// TIA Portal V17 export
// export: Created 2024-09-02T12:49:55.2454988Z, ExportSetting WithDefaults, DisplayName Totally Integrated Automation Portal, DisplayVersion V17, DisplayName TIA Portal Openness, DisplayVersion V17, DisplayName TIA Portal Version Control Interface, DisplayVersion V17, DisplayName STEP 7 Professional, DisplayVersion V17, DisplayName STEP 7 Safety, DisplayVersion V17, DisplayName WinCC Professional, DisplayVersion V17
FUNCTION "SysFC_NumOfElementArray" : Void   // FC129, LAD
TITLE = Determining the number of elements in the array / Anzahl Elemente im Array ermitteln
{ S7_Optimized_Access := 'TRUE' }
AUTHOR : OlegFuehrus
FAMILY : DIAG
NAME : DIAG
VERSION : 0.1
// stored: AutoNumber true, IsIECCheckEnabled false, SetENOAutomatically false, UDAEnableTagReadback false
   VAR_INPUT
      Data : Variant;
   END_VAR
   VAR_OUTPUT
      NumOfElemets : UDInt;
      Fault : Bool;
   END_VAR
   VAR_TEMP
      t_VKE0 : Bool;
      t_VKE1 : Bool;
      t_Amount : UDInt;
      t_Fault : Bool;
   END_VAR
BEGIN

REGION Network 1: VKE0/1
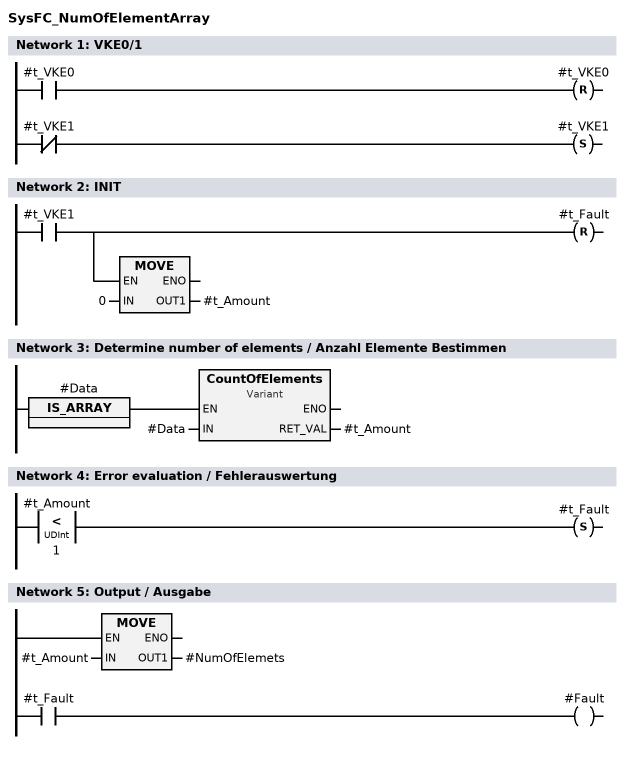
   RUNG wire#powerrail
      Contact( #t_VKE0 )
      R_Coil( #t_VKE0 )
   END_RUNG
   RUNG wire#powerrail
      I_Contact( #t_VKE1 )
      S_Coil( #t_VKE1 )
   END_RUNG
   // the same network as SCL:
   IF #t_VKE0 THEN #t_VKE0 := FALSE; END_IF;
   IF NOT #t_VKE1 THEN #t_VKE1 := TRUE; END_IF;
END_REGION

REGION Network 2: INIT
   RUNG wire#powerrail
      Contact( #t_VKE1 )
      wire#w1
      R_Coil( #t_Fault )
   END_RUNG
   RUNG wire#w1
      Move(in := 0, out1 => #t_Amount)
   END_RUNG
   // the same network as SCL:
   IF #t_VKE1 THEN
       #t_Fault := FALSE;
       #t_Amount := 0;
   END_IF;
END_REGION

REGION Network 3: Determine number of elements / Anzahl Elemente Bestimmen
   // no SCL statement known for CountOfElements, IS_ARRAY: written as a call
   IF IS_ARRAY(#Data) THEN #t_Amount := CountOfElements(in := #Data); END_IF;
END_REGION

REGION Network 4: Error evaluation / Fehlerauswertung
   RUNG wire#powerrail
      { S7_Templates := "SrcType := UDInt" } LT_Contact(in1 := #t_Amount, in2 := 1)
      S_Coil( #t_Fault )
   END_RUNG
   // the same network as SCL:
   IF #t_Amount < 1 THEN #t_Fault := TRUE; END_IF;
END_REGION

REGION Network 5: Output / Ausgabe
   RUNG wire#powerrail
      Move(in := #t_Amount, out1 => #NumOfElemets)
   END_RUNG
   RUNG wire#powerrail
      Contact( #t_Fault )
      Coil( #Fault )
   END_RUNG
   // the same network as SCL:
   #NumOfElemets := #t_Amount;
   #Fault := #t_Fault;
END_REGION
END_FUNCTION
